(* PLC project syrup_weighing, Dassault Systèmes ControlBuild 2024x *)
(* stored: creationDateTime 2023-10-03T11:13:37-01:00 *)

FUNCTION_BLOCK batch.syrup_weighing
  VAR_INPUT
    weighingRequest : BOOL := false;
    cycleInProgress : BOOL := false;
    weighingWeight : DINT := 0;
  END_VAR
  VAR_INPUT
    syrup1Weight : DINT := 0;
    syrup2Weight : DINT := 0;
    syrup3Weight : DINT := 0;
  END_VAR
  VAR_OUTPUT
    weighingOk : BOOL := false;
  END_VAR
  VAR_OUTPUT
    introduceS1 : BOOL := false;
    introS1End : BOOL := false;
  END_VAR
  VAR_OUTPUT
    introduceS2 : BOOL := false;
    introS2End : BOOL := false;
  END_VAR
  VAR_OUTPUT
    introduceS3 : BOOL := false;
    introS3End : BOOL := false;
  END_VAR
  VAR_OUTPUT
    exitSyrup : BOOL := false;
    exitSyrupEnd : BOOL := false;
  END_VAR
  VAR
    totalWeight : DINT := 0;
    weighingS1 : BOOL := false;
    weighingS2 : BOOL := false;
    weighingS3 : BOOL := false;
    weighingS1Ok : BOOL := false;
    weighingS2Ok : BOOL := false;
    weighingS3Ok : BOOL := false;
    endOfWeighingS3 : BOOL := false;
    endOfWeighingS2 : BOOL := false;
    endOfWeighingS1 : BOOL := false;
  END_VAR
  VAR CONSTANT
    maxWeight : DINT := 200;
  END_VAR

INITIAL_STEP 10:
  COMPUTE_FUNCTION_BLOCKS(S);
END_STEP
TRANSITION FROM 10 TO 11
  := weighingS1;
END_TRANSITION
INITIAL_STEP 20:
END_STEP
TRANSITION FROM 20 TO 21
  := cycleInProgress AND weighingRequest;
END_TRANSITION
INITIAL_STEP 30:
END_STEP
TRANSITION FROM 30 TO 31
  := weighingS2;
END_TRANSITION
INITIAL_STEP 40:
END_STEP
TRANSITION FROM 40 TO 41
  := weighingS3;
END_TRANSITION
STEP 11:
  11_INLINE1(N);
END_STEP
ACTION 11_INLINE1:
  introduceS1;
END_ACTION
TRANSITION FROM 11 TO 12
  := endOfWeighingS1;
END_TRANSITION
STEP 21:
  21_INLINE2(N);
END_STEP
ACTION 21_INLINE2:
  IF (syrup1Weight > 0) THEN
  	weighingS1;
  END_IF;
END_ACTION
TRANSITION FROM 21 TO 22
  := cycleInProgress AND (weighingS1Ok OR (syrup1Weight <= 0));
END_TRANSITION
STEP 12:
  12_INLINE3(N);
END_STEP
ACTION 12_INLINE3:
  IF(RE X12) THEN
  	totalWeight := totalWeight + weighingWeight;
  END_IF;
END_ACTION
TRANSITION FROM 12 TO 13
  := cycleInProgress AND T/X12/250ms;
END_TRANSITION
STEP 22:
  22_INLINE4(N);
END_STEP
ACTION 22_INLINE4:
  IF (syrup2Weight > 0) THEN
  	weighingS2;
  END_IF;
END_ACTION
TRANSITION FROM 22 TO 23
  := cycleInProgress AND (weighingS2Ok OR (syrup2Weight <= 0));
END_TRANSITION
STEP 13:
  13_INLINE5(N);
END_STEP
ACTION 13_INLINE5:
  exitSyrup;
END_ACTION
TRANSITION FROM 13 TO 14
  := weighingWeight <= 1;
END_TRANSITION
STEP 23:
  23_INLINE6(N);
END_STEP
ACTION 23_INLINE6:
  IF (syrup3Weight > 0) THEN
  	weighingS3;
  END_IF;
END_ACTION
TRANSITION FROM 23 TO 24
  := cycleInProgress AND (weighingS3Ok OR (syrup3Weight <= 0));
END_TRANSITION
STEP 14:
END_STEP
TRANSITION FROM 14 TO 15
  := cycleInProgress AND (totalWeight >= syrup1Weight);
END_TRANSITION
TRANSITION FROM 14 TO 11
  := cycleInProgress AND (totalWeight < syrup1Weight);
END_TRANSITION
STEP 24:
  24_INLINE7(N);
END_STEP
ACTION 24_INLINE7:
  weighingOk;
END_ACTION
TRANSITION FROM 24 TO 20
  := NOT weighingRequest;
END_TRANSITION
STEP 15:
  15_INLINE8(N);
END_STEP
ACTION 15_INLINE8:
  weighingS1Ok;
  totalWeight := 0;
END_ACTION
TRANSITION FROM 15 TO 10
  := NOT weighingS1;
END_TRANSITION
STEP 31:
  31_INLINE9(N);
END_STEP
ACTION 31_INLINE9:
  introduceS2;
END_ACTION
TRANSITION FROM 31 TO 32
  := endOfWeighingS2;
END_TRANSITION
STEP 41:
  41_INLINE10(N);
END_STEP
ACTION 41_INLINE10:
  introduceS3;
END_ACTION
TRANSITION FROM 41 TO 42
  := endOfWeighingS3;
END_TRANSITION
STEP 32:
  32_INLINE11(N);
END_STEP
ACTION 32_INLINE11:
  IF(RE X32) THEN
  	totalWeight := totalWeight + weighingWeight;
  END_IF;
END_ACTION
TRANSITION FROM 32 TO 33
  := cycleInProgress AND T/X32/250ms;
END_TRANSITION
STEP 42:
  42_INLINE12(N);
END_STEP
ACTION 42_INLINE12:
  IF(RE X42) THEN
  	totalWeight := totalWeight + weighingWeight;
  END_IF;
END_ACTION
TRANSITION FROM 42 TO 43
  := cycleInProgress AND T/X42/250ms;
END_TRANSITION
STEP 33:
  33_INLINE13(N);
END_STEP
ACTION 33_INLINE13:
  exitSyrup;
END_ACTION
TRANSITION FROM 33 TO 34
  := weighingWeight<=1;
END_TRANSITION
STEP 43:
  43_INLINE14(N);
END_STEP
ACTION 43_INLINE14:
  exitSyrup;
END_ACTION
TRANSITION FROM 43 TO 44
  := weighingWeight<=1;
END_TRANSITION
STEP 44:
END_STEP
TRANSITION FROM 44 TO 45
  := cycleInProgress AND (totalWeight >= syrup3Weight);
END_TRANSITION
TRANSITION FROM 44 TO 41
  := cycleInProgress AND (totalWeight < syrup3Weight);
END_TRANSITION
STEP 34:
END_STEP
TRANSITION FROM 34 TO 35
  := cycleInProgress AND (totalWeight >= syrup2Weight);
END_TRANSITION
TRANSITION FROM 34 TO 31
  := cycleInProgress AND (totalWeight < syrup2Weight);
END_TRANSITION
STEP 45:
  45_INLINE15(N);
END_STEP
ACTION 45_INLINE15:
  weighingS3Ok;
  totalWeight := 0;
END_ACTION
TRANSITION FROM 45 TO 40
  := NOT weighingS3;
END_TRANSITION
STEP 35:
  35_INLINE16(N);
END_STEP
ACTION 35_INLINE16:
  weighingS2Ok;
  totalWeight := 0;
END_ACTION
TRANSITION FROM 35 TO 30
  := NOT weighingS2;
END_TRANSITION
ACTION COMPUTE_FUNCTION_BLOCKS:  (* blocks drawn on the SFC sheet *)
  G1:
  G2:
  G3:
  G4:
END_ACTION

ACTION PreSFC:
endOfWeighingS1 := ((totalWeight + weighingWeight) >= syrup1Weight) OR (weighingWeight >= maxWeight);
endOfWeighingS2 := ((totalWeight + weighingWeight) >= syrup2Weight) OR (weighingWeight >= maxWeight);
endOfWeighingS3 := ((totalWeight + weighingWeight) >= syrup3Weight) OR (weighingWeight >= maxWeight);
END_ACTION

ACTION PostSFC:
IF NOT cycleInProgress THEN
	introduceS1 := FALSE;
	introduceS2 := FALSE;
	introduceS3 := FALSE;
	exitSyrup := FALSE;
END_IF;

introS1End := NOT cycleInProgress OR NOT introduceS1;
introS2End := NOT cycleInProgress OR NOT introduceS2;
introS3End := NOT cycleInProgress OR NOT introduceS3;
exitSyrupEnd := NOT cycleInProgress OR NOT exitSyrup;
END_ACTION
END_FUNCTION_BLOCK
